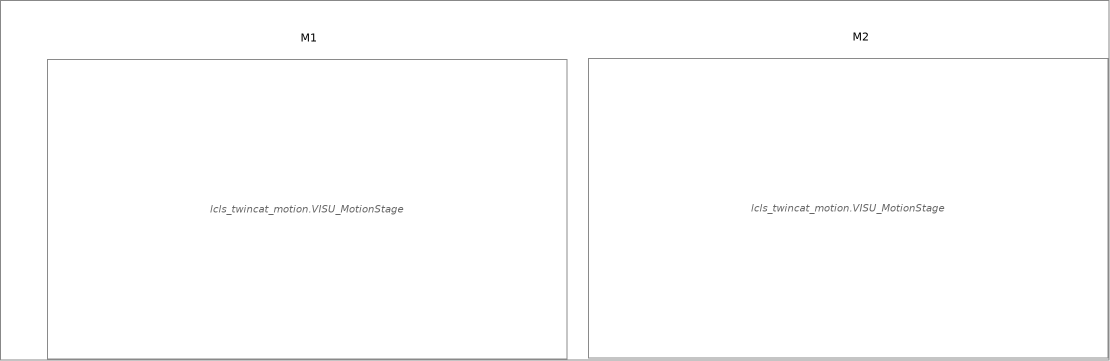
VISUALIZATION Visualization  // 1110x361
    Frame (47,59 520x300)
        shows lcls_twincat_motion.VISU_MotionStage(VisuMotionStage := Main.M1)
    Frame (588,58 520x300)
        shows lcls_twincat_motion.VISU_MotionStage(VisuMotionStage := Main.M2)
    Label (786,22 150x30), "M2"
    Label (234,23 150x30), "M1"
END_VISUALIZATION

(* stored: Version 1.1.0.1, ProductVersion 3.1.4022.12
   Visu Visualization: Id {76b5adfc-173c-4e5d-abbf-10e21d66f08b} *)
